FUNCTION_BLOCK ADI_FB_CTU (* Up counter (DINT) ADI-Adapter Version *)
  (* Standard: 61499-2; Description: Copyright (c) 2026 Meisterschulen am Ostbahnhof This program and the accompanying materials are made available under the terms of the Eclipse Public License 2.0 which is available at https://www.eclipse.org/legal/epl-2.0/ SPDX-License-Identifier: EPL-2.0 NOTE: This block fires the AX output event (Q.E1) on every update (CU, R, PV). If on-change triggering is required, use of an AX_D_FF as a filter is recommended. *)
  (* Version 1.0, 2026-04-21, Franz Höpfinger, Meisterschulen am Ostbahnhof, initial API and implementation and/or initial documentation *)
  PACKAGE adapter::iec61131::counters;
  IMPORT eclipse4diac::core::TypeHash;
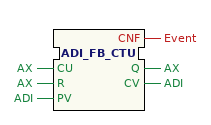
  EVENT_OUTPUT
    CNF; (* Execution Confirmation *)
  END_EVENT
  SOCKETS
    CU : adapter::types::unidirectional::AX; (* Count up *)
    R : adapter::types::unidirectional::AX; (* Reset *)
    PV : adapter::types::unidirectional::ADI; (* Preset value *)
  END_SOCKETS
  PLUGS
    Q : adapter::types::unidirectional::AX; (* Output *)
    CV : adapter::types::unidirectional::ADI; (* Count value *)
  END_PLUGS
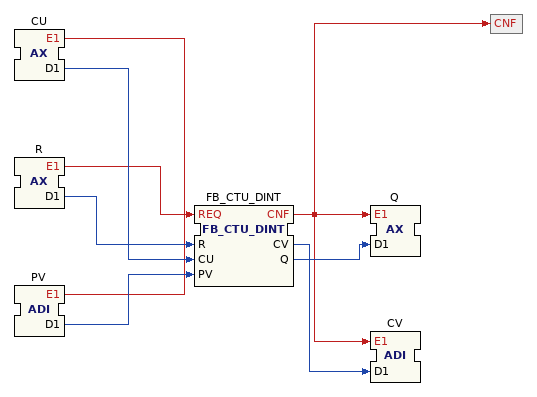
  FBS
    FB_CTU_DINT : iec61131::counters::FB_CTU_DINT;
  END_FBS
  EVENT_CONNECTIONS
    R.E1 TO FB_CTU_DINT.REQ;
    CU.E1 TO FB_CTU_DINT.REQ;
    PV.E1 TO FB_CTU_DINT.REQ;
    FB_CTU_DINT.CNF TO CV.E1;
    FB_CTU_DINT.CNF TO Q.E1;
    FB_CTU_DINT.CNF TO CNF;
  END_CONNECTIONS
  DATA_CONNECTIONS
    R.D1 TO FB_CTU_DINT.R;
    CU.D1 TO FB_CTU_DINT.CU;
    PV.D1 TO FB_CTU_DINT.PV;
    FB_CTU_DINT.CV TO CV.D1;
    FB_CTU_DINT.Q TO Q.D1;
  END_CONNECTIONS
END_FUNCTION_BLOCK
